// TwinCAT 3 PLC project State_Pattern
// ProgramVersion: 3.1.4024.0
// libraries:
//   Tc2_Standard, * (Beckhoff Automation GmbH)
//   Tc2_System, * (Beckhoff Automation GmbH)
//   Tc3_Module, * (Beckhoff Automation GmbH)
// project tree:
//   PackML States/Idle/ Aborted.TcPOU, Execute.TcPOU, Idle.TcPOU, Stopped.TcPOU
//   PackML States/ ITF_States.TcIO, ITF_PackMLState.TcIO
//   PackML States/Transition/ Aborting.TcPOU, Clearing.TcPOU, Resetting.TcPOU, Starting.TcPOU, Stopping.TcPOU
//   PackML/ ITF_PackMLMachine.TcIO, SomeMachine.TcPOU
//   / PlcTask.TcTTO
//   POUs/ MAIN.TcPOU
// (motion and I/O tree: see PLC project simple_factory_pattern)
// real-time tasks:
//   TASK PlcTask: cycle T#10ms, priority 20, ADS port 350
//   TASK PlcTask1: cycle T#10ms, priority 21, ADS port 351
//   TASK PlcTask2: cycle T#10ms, priority 22, ADS port 352
//   TASK PlcTask3: cycle T#10ms, priority 23, ADS port 353
//   TASK PlcTask4: cycle T#10ms, priority 24, ADS port 354
//   TASK PlcTask5: cycle T#10ms, priority 25, ADS port 355
//   TASK PlcTask6: cycle T#10ms, priority 26, ADS port 356
//   TASK PlcTask7: cycle T#10ms, priority 27, ADS port 357
//   TASK PlcTask8: cycle T#10ms, priority 28, ADS port 358
//   TASK PlcTask9: cycle T#10ms, priority 29, ADS port 359
//   TASK PlcTask10: cycle T#10ms, priority 30, ADS port 360
//   TASK PlcTask11: cycle T#10ms, priority 31, ADS port 361

CONFIGURATION State_Pattern
    RESOURCE PLC ON TwinCAT3
        TASK PlcTask(INTERVAL := T#10ms, PRIORITY := 25);
        PROGRAM MAIN WITH PlcTask : MAIN;
    END_RESOURCE
END_CONFIGURATION

// ---- PackML States/ITF_States.TcIO
INTERFACE ITF_States

PROPERTY AbortingState : ITF_PackMLState
GET
END_GET
SET
END_SET
END_PROPERTY

PROPERTY MyNextState : ITF_PackMLState
GET
END_GET
SET
END_SET
END_PROPERTY

PROPERTY StoppingState : ITF_PackMLState
GET
END_GET
SET
END_SET
END_PROPERTY

END_INTERFACE

// ---- PackML/ITF_PackMLMachine.TcIO
INTERFACE ITF_PackMLMachine

METHOD ChangeState : BOOL
VAR_INPUT
	NewState : ITF_PackMLState;
END_VAR
END_METHOD

END_INTERFACE

// ---- PackML States/ITF_PackMLState.TcIO
INTERFACE ITF_PackMLState

METHOD CyclicLogic : BOOL
VAR_INPUT
END_VAR
END_METHOD

METHOD EStop : BOOL
VAR_INPUT
END_VAR
END_METHOD

METHOD Reset : BOOL
VAR_INPUT
END_VAR
END_METHOD

METHOD SetContext : BOOL
VAR_INPUT
	context : ITF_PackMLMachine;
END_VAR
END_METHOD

METHOD Start : BOOL
VAR_INPUT
END_VAR
END_METHOD

METHOD Stop : BOOL
VAR_INPUT
END_VAR
END_METHOD

END_INTERFACE

// ---- POUs/MAIN.TcPOU
PROGRAM MAIN
VAR
	MyMachine : SomeMachine;
	HMIStartButton : BOOL;
	HMIResetButton : BOOL;
	HMIStopButton : BOOL;
	ESTOP : BOOL;
END_VAR

MyMachine.CyclicLogic();

IF HMIStartButton THEN
	HMIStartButton := FALSE;
	MyMachine.Start();
END_IF

IF HMIStopButton THEN
	HMIStopButton := FALSE;
	MyMachine.Stop();
END_IF

IF HMIResetButton THEN
	HMIResetButton := FALSE;
	MyMachine.Reset();
END_IF

IF ESTOP THEN
	ESTOP := FALSE;
	MyMachine.EStop();
END_IF

END_PROGRAM

// ---- PackML/SomeMachine.TcPOU
FUNCTION_BLOCK SomeMachine IMPLEMENTS ITF_PackMLMachine
VAR
	_MyState : ITF_PackMLState;
	_Aborting : Aborting := (MyNextState := _Aborted);
	_Aborted : Aborted := (MyNextState := _Clearing);
	_Clearing : Clearing := (MyNextState := _Stopped);
	_Stopped : Stopped;
END_VAR

METHOD ChangeState : BOOL
VAR_INPUT
	NewState : ITF_PackMLState;
END_VAR
_MyState := NewState;
_MyState.SetContext(this^);
END_METHOD

METHOD CyclicLogic : BOOL
VAR_INPUT
END_VAR
IF _MyState <> 0 THEN
	_MyState.CyclicLogic();
END_IF
END_METHOD

METHOD EStop : BOOL
VAR_INPUT
END_VAR
IF _MyState <> 0 THEN
	_MyState.EStop();
END_IF
END_METHOD

METHOD Reset : BOOL
VAR_INPUT
END_VAR
IF _MyState <> 0 THEN
	_MyState.Reset();
END_IF
END_METHOD

METHOD Start : BOOL
VAR_INPUT
END_VAR
IF _MyState <> 0 THEN
	_MyState.Start();
END_IF
END_METHOD

METHOD Stop : BOOL
VAR_INPUT
END_VAR
IF _MyState <> 0 THEN
	_MyState.Stop();
END_IF
END_METHOD

END_FUNCTION_BLOCK

// ---- PackML States/Transition/Aborting.TcPOU
FUNCTION_BLOCK Aborting IMPLEMENTS ITF_PackMLState, ITF_States
VAR
	_MyContext : ITF_PackMLMachine;
END_VAR

{warning 'add property implementation'}
PROPERTY AbortingState : ITF_PackMLState
GET
END_GET
SET
END_SET
END_PROPERTY

METHOD CyclicLogic : BOOL
VAR_INPUT
END_VAR
END_METHOD

{warning 'add method implementation '}
METHOD EStop : BOOL
END_METHOD

{warning 'add property implementation'}
PROPERTY MyNextState : ITF_PackMLState
GET
END_GET
SET
END_SET
END_PROPERTY

{warning 'add method implementation '}
METHOD Reset : BOOL
END_METHOD

METHOD SetContext : BOOL
VAR_INPUT
	context	: ITF_PackMLMachine;
END_VAR
_MyContext := context;
END_METHOD

{warning 'add method implementation '}
METHOD Start : BOOL
END_METHOD

{warning 'add method implementation '}
METHOD Stop : BOOL
END_METHOD

{warning 'add property implementation'}
PROPERTY StoppingState : ITF_PackMLState
GET
END_GET
SET
END_SET
END_PROPERTY

END_FUNCTION_BLOCK

// ---- PackML States/Idle/Aborted.TcPOU
FUNCTION_BLOCK Aborted IMPLEMENTS ITF_PackMLState, ITF_States
VAR
	_MyContext : ITF_PackMLMachine;
END_VAR

{warning 'add property implementation'}
PROPERTY AbortingState : ITF_PackMLState
GET
END_GET
SET
END_SET
END_PROPERTY

METHOD CyclicLogic : BOOL
VAR_INPUT
END_VAR
END_METHOD

{warning 'add method implementation '}
METHOD EStop : BOOL
END_METHOD

{warning 'add property implementation'}
PROPERTY MyNextState : ITF_PackMLState
GET
END_GET
SET
END_SET
END_PROPERTY

{warning 'add method implementation '}
METHOD Reset : BOOL
END_METHOD

METHOD SetContext : BOOL
VAR_INPUT
	context	: ITF_PackMLMachine;
END_VAR
_MyContext := context;
END_METHOD

{warning 'add method implementation '}
METHOD Start : BOOL
END_METHOD

{warning 'add method implementation '}
METHOD Stop : BOOL
END_METHOD

{warning 'add property implementation'}
PROPERTY StoppingState : ITF_PackMLState
GET
END_GET
SET
END_SET
END_PROPERTY

END_FUNCTION_BLOCK

// ---- PackML States/Transition/Clearing.TcPOU
FUNCTION_BLOCK Clearing IMPLEMENTS ITF_PackMLState, ITF_States
VAR
	_MyContext : ITF_PackMLMachine;
END_VAR

{warning 'add property implementation'}
PROPERTY AbortingState : ITF_PackMLState
GET
END_GET
SET
END_SET
END_PROPERTY

METHOD CyclicLogic : BOOL
VAR_INPUT
END_VAR
END_METHOD

{warning 'add method implementation '}
METHOD EStop : BOOL
END_METHOD

{warning 'add property implementation'}
PROPERTY MyNextState : ITF_PackMLState
GET
END_GET
SET
END_SET
END_PROPERTY

{warning 'add method implementation '}
METHOD Reset : BOOL
END_METHOD

METHOD SetContext : BOOL
VAR_INPUT
	context	: ITF_PackMLMachine;
END_VAR
_MyContext := context;
END_METHOD

{warning 'add method implementation '}
METHOD Start : BOOL
END_METHOD

{warning 'add method implementation '}
METHOD Stop : BOOL
END_METHOD

{warning 'add property implementation'}
PROPERTY StoppingState : ITF_PackMLState
GET
END_GET
SET
END_SET
END_PROPERTY

END_FUNCTION_BLOCK

// ---- PackML States/Idle/Stopped.TcPOU
FUNCTION_BLOCK Stopped IMPLEMENTS ITF_PackMLState, ITF_States
VAR
	_MyContext : ITF_PackMLMachine;
END_VAR

{warning 'add property implementation'}
PROPERTY AbortingState : ITF_PackMLState
GET
END_GET
SET
END_SET
END_PROPERTY

METHOD CyclicLogic : BOOL
VAR_INPUT
END_VAR
END_METHOD

{warning 'add method implementation '}
METHOD EStop : BOOL
END_METHOD

{warning 'add property implementation'}
PROPERTY MyNextState : ITF_PackMLState
GET
END_GET
SET
END_SET
END_PROPERTY

{warning 'add method implementation '}
METHOD Reset : BOOL
END_METHOD

{warning 'add method implementation '}
METHOD SetContext : BOOL
VAR_INPUT
	context	: ITF_PackMLMachine;
END_VAR
_MyContext := context;
END_METHOD

{warning 'add method implementation '}
METHOD Start : BOOL
END_METHOD

{warning 'add method implementation '}
METHOD Stop : BOOL
END_METHOD

{warning 'add property implementation'}
PROPERTY StoppingState : ITF_PackMLState
GET
END_GET
SET
END_SET
END_PROPERTY

END_FUNCTION_BLOCK

// ---- PackML States/Idle/Execute.TcPOU
FUNCTION_BLOCK Execute IMPLEMENTS ITF_PackMLState, ITF_States
VAR
	_MyContext : ITF_PackMLMachine;
END_VAR

{warning 'add property implementation'}
PROPERTY AbortingState : ITF_PackMLState
GET
END_GET
SET
END_SET
END_PROPERTY

METHOD CyclicLogic : BOOL
VAR_INPUT
END_VAR
END_METHOD

{warning 'add method implementation '}
METHOD EStop : BOOL
END_METHOD

{warning 'add property implementation'}
PROPERTY MyNextState : ITF_PackMLState
GET
END_GET
SET
END_SET
END_PROPERTY

{warning 'add method implementation '}
METHOD Reset : BOOL
END_METHOD

{warning 'add method implementation '}
METHOD SetContext : BOOL
VAR_INPUT
	context	: ITF_PackMLMachine;
END_VAR
_MyContext := context;
END_METHOD

{warning 'add method implementation '}
METHOD Start : BOOL
END_METHOD

{warning 'add method implementation '}
METHOD Stop : BOOL
END_METHOD

{warning 'add property implementation'}
PROPERTY StoppingState : ITF_PackMLState
GET
END_GET
SET
END_SET
END_PROPERTY

END_FUNCTION_BLOCK

// ---- PackML States/Idle/Idle.TcPOU
FUNCTION_BLOCK Idle IMPLEMENTS ITF_PackMLState, ITF_States
VAR
	_MyContext : ITF_PackMLMachine;
END_VAR

{warning 'add property implementation'}
PROPERTY AbortingState : ITF_PackMLState
GET
END_GET
SET
END_SET
END_PROPERTY

METHOD CyclicLogic : BOOL
VAR_INPUT
END_VAR
END_METHOD

{warning 'add method implementation '}
METHOD EStop : BOOL
END_METHOD

{warning 'add property implementation'}
PROPERTY MyNextState : ITF_PackMLState
GET
END_GET
SET
END_SET
END_PROPERTY

{warning 'add method implementation '}
METHOD Reset : BOOL
END_METHOD

{warning 'add method implementation '}
METHOD SetContext : BOOL
VAR_INPUT
	context	: ITF_PackMLMachine;
END_VAR
_MyContext := context;
END_METHOD

{warning 'add method implementation '}
METHOD Start : BOOL
END_METHOD

{warning 'add method implementation '}
METHOD Stop : BOOL
END_METHOD

{warning 'add property implementation'}
PROPERTY StoppingState : ITF_PackMLState
GET
END_GET
SET
END_SET
END_PROPERTY

END_FUNCTION_BLOCK

// ---- PackML States/Transition/Resetting.TcPOU
FUNCTION_BLOCK Resetting IMPLEMENTS ITF_PackMLState, ITF_States
VAR
	_MyContext : ITF_PackMLMachine;
END_VAR

{warning 'add property implementation'}
PROPERTY AbortingState : ITF_PackMLState
GET
END_GET
SET
END_SET
END_PROPERTY

METHOD CyclicLogic : BOOL
VAR_INPUT
END_VAR
END_METHOD

{warning 'add method implementation '}
METHOD EStop : BOOL
END_METHOD

{warning 'add property implementation'}
PROPERTY MyNextState : ITF_PackMLState
GET
END_GET
SET
END_SET
END_PROPERTY

{warning 'add method implementation '}
METHOD Reset : BOOL
END_METHOD

METHOD SetContext : BOOL
VAR_INPUT
	context	: ITF_PackMLMachine;
END_VAR
_MyContext := context;
END_METHOD

{warning 'add method implementation '}
METHOD Start : BOOL
END_METHOD

{warning 'add method implementation '}
METHOD Stop : BOOL
END_METHOD

{warning 'add property implementation'}
PROPERTY StoppingState : ITF_PackMLState
GET
END_GET
SET
END_SET
END_PROPERTY

END_FUNCTION_BLOCK

// ---- PackML States/Transition/Starting.TcPOU
FUNCTION_BLOCK Starting IMPLEMENTS ITF_PackMLState, ITF_States
VAR
	_MyContext : ITF_PackMLMachine;
END_VAR

{warning 'add property implementation'}
PROPERTY AbortingState : ITF_PackMLState
GET
END_GET
SET
END_SET
END_PROPERTY

METHOD CyclicLogic : BOOL
VAR_INPUT
END_VAR
END_METHOD

{warning 'add method implementation '}
METHOD EStop : BOOL
END_METHOD

{warning 'add property implementation'}
PROPERTY MyNextState : ITF_PackMLState
GET
END_GET
SET
END_SET
END_PROPERTY

{warning 'add method implementation '}
METHOD Reset : BOOL
END_METHOD

METHOD SetContext : BOOL
VAR_INPUT
	context	: ITF_PackMLMachine;
END_VAR
_MyContext := context;
END_METHOD

{warning 'add method implementation '}
METHOD Start : BOOL
END_METHOD

{warning 'add method implementation '}
METHOD Stop : BOOL
END_METHOD

{warning 'add property implementation'}
PROPERTY StoppingState : ITF_PackMLState
GET
END_GET
SET
END_SET
END_PROPERTY

END_FUNCTION_BLOCK

// ---- PackML States/Transition/Stopping.TcPOU
FUNCTION_BLOCK Stopping IMPLEMENTS ITF_PackMLState, ITF_States
VAR
	_MyContext : ITF_PackMLMachine;
END_VAR

{warning 'add property implementation'}
PROPERTY AbortingState : ITF_PackMLState
GET
END_GET
SET
END_SET
END_PROPERTY

METHOD CyclicLogic : BOOL
VAR_INPUT
END_VAR
END_METHOD

{warning 'add method implementation '}
METHOD EStop : BOOL
END_METHOD

{warning 'add property implementation'}
PROPERTY MyNextState : ITF_PackMLState
GET
END_GET
SET
END_SET
END_PROPERTY

{warning 'add method implementation '}
METHOD Reset : BOOL
END_METHOD

METHOD SetContext : BOOL
VAR_INPUT
	context	: ITF_PackMLMachine;
END_VAR
_MyContext := context;
END_METHOD

{warning 'add method implementation '}
METHOD Start : BOOL
END_METHOD

{warning 'add method implementation '}
METHOD Stop : BOOL
END_METHOD

{warning 'add property implementation'}
PROPERTY StoppingState : ITF_PackMLState
GET
END_GET
SET
END_SET
END_PROPERTY

END_FUNCTION_BLOCK
